{attribute 'qualified_only'}
{attribute 'strict'}
TYPE E_SubElement_Types :
(
	No 						:= 0,
	
	With_fix_subelements	:= 1,
	With_list 				:= 2,
	
	Fix_subelement			:= 17,	
	List_element			:= 18
) BYTE;
END_TYPE

(* stored: Version 1.1.0.1, ProductVersion 3.1.4024.11
   DUT E_SubElement_Types: Id {1443e881-0bc3-4e51-a57b-e72a684a99fb} *)
